PROGRAM PRG_OpslagFoutDetectie
VAR
	SensorHoog		AT		%I*		:BOOL;
	SensorLaag		AT		%I*		:BOOL;
	StartKnop		AT		%I*		:BOOL;
	StopKnop		AT		%I*		:BOOL;
	
	Klep			AT		%Q*		:BOOL;
	Pomp			AT		%Q*		:BOOL;
	Vullen			AT		%Q*		:BOOL;
END_VAR

Klep := SensorLaag AND NOT(SensorHoog);
Vullen := SensorLaag AND NOT(SensorHoog);

IF StopKnop OR Vullen OR NOT(SensorLaag) OR (SensorLaag AND NOT(SensorHoog)) OR NOT(StartKnop) THEN
	Pomp := FALSE;
ELSIF StartKnop THEN
	Pomp := TRUE; 
END_IF

END_PROGRAM

(* stored: Version 1.1.0.1, ProductVersion 3.1.4024.15
   POU PRG_OpslagFoutDetectie: Id {f6aa53c6-2d27-467c-ac67-f01685315add}, SpecialFunc None *)
